PROGRAM PRG_IM4K2_PPM
VAR
    {attribute 'pytmc' := 'pv: IM4K2:PPM'}
    {attribute 'TcLinkTo' := '.fbGige.iIlluminatorINT := TIIB[IM4K2-EL4004-E7]^AO Outputs Channel 1^Analog output;
                              .fbGige.bGigePower := TIIB[IM4K2-EL2004-E3]^Channel 2^Output;
                              .fbPowerMeter.iVoltageINT := TIIB[IM4K2-EL3602-0002-E8]^AI Inputs Channel 1^Value;
                              .fbPowerMeter.fbTempSensor.bError := TIIB[IM4K2-EL3314-E4]^TC Inputs Channel 1^Status^Error;
                              .fbPowerMeter.fbTempSensor.bUnderrange := TIIB[IM4K2-EL3314-E4]^TC Inputs Channel 1^Status^Underrange;
                              .fbPowerMeter.fbTempSensor.bOverrange := TIIB[IM4K2-EL3314-E4]^TC Inputs Channel 1^Status^Overrange;
                              .fbPowerMeter.fbTempSensor.iRaw := TIIB[IM4K2-EL3314-E4]^TC Inputs Channel 1^Value;
                              .fbYagTempSensor.bError := TIIB[IM4K2-EL3314-E4]^TC Inputs Channel 2^Status^Error;
                              .fbYagTempSensor.bUnderrange := TIIB[IM4K2-EL3314-E4]^TC Inputs Channel 2^Status^Underrange;
                              .fbYagTempSensor.bOverrange := TIIB[IM4K2-EL3314-E4]^TC Inputs Channel 2^Status^Overrange;
                              .fbYagTempSensor.iRaw := TIIB[IM4K2-EL3314-E4]^TC Inputs Channel 2^Value;
                              .fbFlowMeter.iRaw := TIIB[IM1K2-EL3052-E5]^AI Standard Channel 1^Value'}
// IM4K2 shares the same flow meter as IM1K2
    fbIM4K2: FB_PPM;

    fbStateSetup: FB_StateSetupHelper;
    stDefault: ST_PositionState := (
        fVelocity := 12,
        bMoveOk := TRUE,
        bValid := TRUE
    );
END_VAR


fbStateSetup(stPositionState:=stDefault, bSetDefault:=TRUE);

fbStateSetup(stPositionState:=fbIM4K2.stOut, fPosition:=-10.80, sPmpsState:='IM4K2:PPM-OUT');
fbStateSetup(stPositionState:=fbIM4K2.stPower, fPosition:=-49.90, sPmpsState:='IM4K2:PPM-POWERMETER');
fbStateSetup(stPositionState:=fbIM4K2.stYag1, fPosition:=-73.90, sPmpsState:='IM4K2:PPM-YAG1');
fbStateSetup(stPositionState:=fbIM4K2.stYag2, fPosition:=-99.91, sPmpsState:='IM4K2:PPM-YAG2');

fbIM4K2(
    fbFFHWO := GVL.fbFastFaultOutput2,
    fbArbiter := GVL.fbArbiter2,
    stYStage := Main.M8,
    sDeviceName := 'IM4K2:PPM',
    sTransitionKey := 'IM4K2:PPM-TRANSITION',
    bEnableMotion := TRUE,
    bEnableBeamParams := TRUE,
    bEnablePositionLimits := TRUE,
    fResponsivity := 0.0584,
    iTermBits := 31,
    fTermMax := 0.2,
    fTermMin := -0.2,
);

END_PROGRAM

(* stored: Version 1.1.0.1, ProductVersion 3.1.4024.12
   POU PRG_IM4K2_PPM: Id {dfd57a27-7901-4447-85ac-e5255b9203c4}, SpecialFunc None *)
